FUNCTION_BLOCK FB_BinarySensor EXTENDS FB_SensorBase
VAR_INPUT
END_VAR
VAR_OUTPUT
END_VAR
VAR
END_VAR

METHOD HandleMessage : BOOL
VAR_INPUT
	message :STRING;
END_VAR
IF message='1' THEN
	ADSLOGSTR(msgCtrlMask := ADSLOG_MSGTYPE_ERROR, msgFmtStr := 'Door Opened', strArg := '');
END_IF
END_METHOD

END_FUNCTION_BLOCK

(* stored: Version 1.1.0.1, ProductVersion 3.1.4024.9
   POU FB_BinarySensor: Id {89e1e01f-36dd-4a6d-bc09-97732e6d9a41}, SpecialFunc None
   Method HandleMessage: Id {2a5c1ba4-da33-45bc-b2dd-dd45456c17bf} *)
